{attribute 'qualified_only'}
VAR_GLOBAL
    Robot1 : TcoAbbRobotics.TcoIrc5_IO_v_1_x_x;
    Robot2 : TcoAbbRobotics.TcoOmnicore_IO_v_1_x_x;
END_VAR

(* stored: Version 1.1.0.1, ProductVersion 3.1.4024.12
   GVL GVL: Id {79f8c6f8-f04d-039b-25af-d31339b2bdfa} *)
